% RSLogix 500 project PLC_1_L4-1.RSS, saved by version 12.00.00.00 %
PROJECT "UNTITLED"    % processor: Bul.1763 MicroLogix 1100 Series B %

PROGRAM FILES
  LAD 2   2 rungs

DATA FILES
  O0 OUTPUT  5 elements
  I1 INPUT  6 elements
  S2 STATUS  66 elements
  B3 BINARY  1 elements
  T4 TIMER  1 elements
  C5 COUNTER  1 elements
  R6 CONTROL  1 elements
  N7 INTEGER  1 elements
  F8 FLOAT  1 elements

LADDER 2
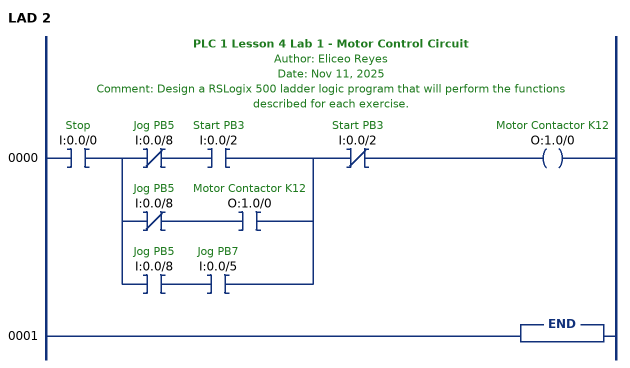
% Rung: 0 %
% TITLE: PLC 1 Lesson 4 Lab 1 - Motor Control Circuit %
% Author: Eliceo Reyes
% Date: Nov 11, 2025
% Comment: Design a RSLogix 500 ladder logic program that will perform the functions described for each exercise. %
SOR XIC I:0.0/0 BST XIO I:0.0/8 XIC I:0.0/2 NXB XIO I:0.0/8 XIC O:1.0/0 NXB XIC I:0.0/8 XIC I:0.0/5 BND XIO I:0.0/2 OTE O:1.0/0 EOR
%   I:0.0/0  "Stop" %
%   I:0.0/8  PB5  "Jog" %
%   I:0.0/2  PB3  "Start" %
%   O:1.0/0  K12  "Motor Contactor" %
%   I:0.0/5  PB7  "Jog" %
% Rung: 1 %
SOR END EOR

OTHER DOCUMENTED ADDRESSES
  I:0.0/1  PB2  "Run/Job Selector"
  I:0.0/4  PB4  "Motor Overload"
  I:0.0/6  PB1  "Stop"
  XIC  "Start"
